// TIA Portal project "Pres Tezgahı" (V16)

(* hardware
DEVICE "S71500/ET200MP station_1"  S7-1500 station
   slot 0: "Rail_0"  Rack  6ES7 590-1***0-0AA0
   slot 1: "PLC_1"  CPU 1513-1 PN  6ES7 513-1AL00-0AB0  V1.8
      slot 3: "CPU display_1"  6ES7591-1AA00-0AA0
      slot 32768: "PROFINET interface_1"  X1
         slot 32769: "Port_1"  X1 P1
         slot 32770: "Port_2"  X1 P2
DEVICE "HMI_2"  TP1200 Comfort
   slot 0: "HMI_2"  TP1200 Comfort  6AV2 124-0MC01-0AX0  16.0.0.0
   slot 1: "HMI_RT_2"  TP1200 Comfort  6AV2 124-0MC01-0AX0  16.0.0.0
   slot 5: "HMI_2.IE_CP_1"  PROFINET Interface  16.0.0.0
      slot 1: "PROFINET Interface_1"  PROFINET Interface
         slot 1: "Port_1"  Port
         slot 2: "Port_2"  Port
   slot 7: "HMI_2.MPI/DP_CP_1"  MPI/DP Interface  16.0.0.0
*)

// ===== PLC "PLC_1"  CPU 1513-1 PN =====

VAR_GLOBAL   // PLC tag table "Default tag table"
   "Buton-1" AT %M0.0 : Bool;
   "Buton-2" AT %M0.1 : Bool;
   "Buton-3" AT %M0.2 : Bool;
   "P_TRIG" AT %M0.3 : Bool;
   "Pres" AT %M0.4 : Bool;
   "P_TRIG2" AT %M0.5 : Bool;
   "Pres1" AT %M0.6 : Bool;
END_VAR

ORGANIZATION_BLOCK "Main"   // OB1, LAD, ProgramCycle
TITLE = "Main Program Sweep (Cycle)"
{ S7_Optimized_Access := 'TRUE' }
VERSION : 0.1
   VAR_INPUT
      Initial_Call : Bool;   // Initial call of this OB
      Remanence : Bool;   // =True, if remanent data are available
   END_VAR
   VAR_TEMP   // added for the SCL form of the ladder/FBD networks
      _w1 : Bool;
      _w2 : Bool;
      _w3 : Bool;
      _w4 : Bool;
   END_VAR
BEGIN

REGION Network 1
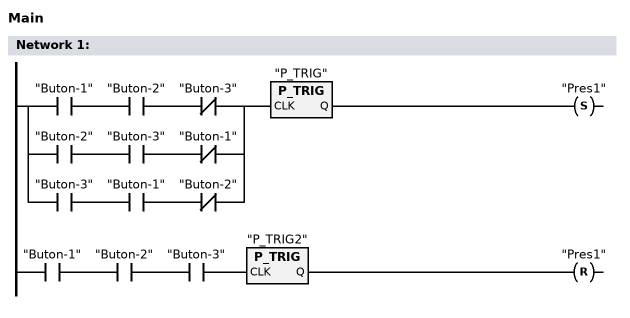
   RUNG wire#powerrail
      Contact( "Buton-1" )
      Contact( "Buton-2" )
      I_Contact( "Buton-3" )
      wire#w1
      P_Trig( "P_TRIG" )
      S_Coil( "Pres1" )
   END_RUNG
   RUNG wire#powerrail
      Contact( "Buton-2" )
      Contact( "Buton-3" )
      I_Contact( "Buton-1" )
   END_RUNG wire#w1
   RUNG wire#powerrail
      Contact( "Buton-3" )
      Contact( "Buton-1" )
      I_Contact( "Buton-2" )
   END_RUNG wire#w1
   RUNG wire#powerrail
      Contact( "Buton-1" )
      Contact( "Buton-2" )
      Contact( "Buton-3" )
      P_Trig( "P_TRIG2" )
      R_Coil( "Pres1" )
   END_RUNG
   // the same network as SCL:
   #_w1 := ("Buton-1" AND "Buton-2" AND NOT "Buton-3") OR ("Buton-2" AND "Buton-3" AND NOT "Buton-1") OR ("Buton-3" AND "Buton-1" AND NOT "Buton-2");
   #_w2 := #_w1 AND NOT "P_TRIG";   // rising edge
   "P_TRIG" := #_w1;
   IF #_w2 THEN "Pres1" := TRUE; END_IF;
   #_w3 := "Buton-1" AND "Buton-2" AND "Buton-3";
   #_w4 := #_w3 AND NOT "P_TRIG2";   // rising edge
   "P_TRIG2" := #_w3;
   IF #_w4 THEN "Pres1" := FALSE; END_IF;
END_REGION
END_ORGANIZATION_BLOCK

(* ===== HMI "HMI_RT_2" =====
system functions are stored by id; their names below are inferred from use

HMI tags "Default tag table"
   "Tag_ScreenNumber" : UInt, internal
   "Buton-1" : Bool = PLC "Buton-1" AT %M0.0
   "Buton-2" : Bool = PLC "Buton-2" AT %M0.1
   "Buton-3" : Bool = PLC "Buton-3" AT %M0.2
   "Pres" : Bool = PLC Pres AT %M0.4
   "Pres1" : Bool = PLC Pres1 AT %M0.6

screen "Root screen" 1280x740, template "Template_1"
   on GenerateScreen: SetTag("Tag_ScreenNumber", 1)
   Button "Button_1" at 211,103 size 96x32; TextOff 'Buton-1'
      on Press: InvertBit("Buton-1")
   Button "Button_2" at 208,160 size 96x32; TextOff 'Buton-2'
      on Press: InvertBit("Buton-2")
   Button "Button_3" at 212,217 size 96x32; TextOff 'Buton-3'
      on Press: InvertBit("Buton-3")

Template "Template_1" 1280x740
   Button "Exit" at 1200,679 size 78x59; TextOff 'Exit'; PictureOff "ExitRuntime_TP1200_Comfort_TR"; PictureOn "ExitRuntime_TP1200_Comfort_TR"
      on Release: StopRuntime(0)
   Button "Template_Button" at 1120,679 size 78x59; TextOff 'Text'
   Button "Template_Button_1" at 1040,679 size 78x59; TextOff 'Text'
   Button "Template_Button_2" at 960,679 size 78x59; TextOff 'Text'
   Button "Template_Button_3" at 880,679 size 78x59; TextOff 'Text'
   Button "Template_Button_4" at 800,679 size 78x59; TextOff 'Text'
   Button "Template_Button_5" at 720,679 size 78x59; TextOff 'Text'
   Button "Template_Button_6" at 640,679 size 78x59; TextOff 'Text'
   Button "Template_Button_7" at 561,679 size 78x59; TextOff 'Text'
   Button "Template_Button_8" at 481,679 size 78x59; TextOff 'Text'
   Button "Template_Button_9" at 401,679 size 78x59; TextOff 'Text'
   Button "Template_Button_10" at 321,679 size 78x59; TextOff 'Text'
   Button "Template_Button_11" at 241,679 size 78x59; TextOff 'Text'
   Button "Template_Button_12" at 161,679 size 78x59; TextOff 'Text'
   Button "Alarms" at 81,679 size 78x59; TextOff 'Alarms'; PictureOff "AlarmDisplay_TP1200_Comfort_TR"; PictureOn "AlarmDisplay_TP1200_Comfort_TR"
      on Release: function_ef3f5d25("Alarm window_Unacknowledged", -1)
   Button "Start screen" at 1,679 size 78x59; TextOff 'Start screen'; PictureOff "NavigateHome_TP1200_Comfort_TR"; PictureOn "NavigateHome_TP1200_Comfort_TR"
      on Release: ActivateScreen("Root screen", 0)
*)